FUNCTION_BLOCK FB_TestString IMPLEMENTS I_BaseString
VAR_INPUT
END_VAR
VAR_OUTPUT
END_VAR
VAR
END_VAR

{warning 'Methodenimplementierung hinzufügen'}
METHOD GetString : STRING
 GetString := 'Test';
END_METHOD

END_FUNCTION_BLOCK

(* stored: Version 1.1.0.1, ProductVersion 3.1.4024.3
   POU FB_TestString: Id {94f83ffd-b2a0-471d-9efa-c5ac1a4418da}, SpecialFunc None
   Method GetString: Id {b893f40f-57b3-4641-a5ef-e802d9c42ccd} *)
